FUNCTION_BLOCK EL6631
VAR
	{attribute addProperty Name "Info data"}
	_infoData : InfoDataAdsAoE;
END_VAR

END_FUNCTION_BLOCK

(* stored: Version 1.1.0.1, ProductVersion 3.1.4024.9
   POU EL6631: Id {ec8ee243-b902-0263-27b9-dcc79375dede}, SpecialFunc None *)
